# EPICS substitutions: apps/snmpApp/Db/gemHV.substitutions
file "db/gemHVcrate.template" {
  pattern { DEV }
          { "HAHV99" }
}
file "db/gemHVchan.template" {
  pattern { DEV, CHAN, Sl, Ch, lolo, low, high, hihi}
          { "HAHV99", "u0", "00", "000", "-50", "-25", "25", "50"}
          { "HAHV99", "u1", "00", "001", "-50", "-25", "25", "50"}
          { "HAHV99", "u2", "00", "002", "-50", "-25", "25", "50"}
          { "HAHV99", "u3", "00", "003", "-50", "-25", "25", "50"}
          { "HAHV99", "u4", "00", "004", "-50", "-25", "25", "50"}
          { "HAHV99", "u5", "00", "005", "-50", "-25", "25", "50"}
          { "HAHV99", "u6", "00", "006", "-50", "-25", "25", "50"}
          { "HAHV99", "u7", "00", "007", "-50", "-25", "25", "50"}
          { "HAHV99", "u100", "01", "000", "-50", "-25", "25", "50"}
          { "HAHV99", "u101", "01", "001", "-50", "-25", "25", "50"}
          { "HAHV99", "u102", "01", "002", "-50", "-25", "25", "50"}
          { "HAHV99", "u103", "01", "003", "-50", "-25", "25", "50"}
          { "HAHV99", "u104", "01", "004", "-50", "-25", "25", "50"}
          { "HAHV99", "u105", "01", "005", "-50", "-25", "25", "50"}
          { "HAHV99", "u106", "01", "006", "-50", "-25", "25", "50"}
          { "HAHV99", "u107", "01", "007", "-50", "-25", "25", "50"}
          { "HAHV99", "u200", "02", "000", "-50", "-25", "25", "50"}
          { "HAHV99", "u201", "02", "001", "-50", "-25", "25", "50"}
          { "HAHV99", "u202", "02", "002", "-50", "-25", "25", "50"}
          { "HAHV99", "u203", "02", "003", "-50", "-25", "25", "50"}
          { "HAHV99", "u204", "02", "004", "-50", "-25", "25", "50"}
          { "HAHV99", "u205", "02", "005", "-50", "-25", "25", "50"}
          { "HAHV99", "u206", "02", "006", "-50", "-25", "25", "50"}
          { "HAHV99", "u207", "02", "007", "-50", "-25", "25", "50"}
}
